{attribute 'qualified_only'}
VAR_GLOBAL
	Section 					: ARRAY[1..4] OF ST_Trip_Base;
	MasterStopPBPressed			: BOOL;
	CaseEStopCircuitBroken		: BOOL;
	ManualModeSelected			: BOOL;
	MCPLossDCpower				: BOOL;
	MCPsystemTripped			: BOOL;
	
	AnyEstopPressed 			: BOOL;
	AllDCpsuOK					: BOOL;
	AnyChargerOverTemp			: BOOL;
	AnyChargerLoadFault			: BOOL;
	AnyChargerInterlockOpen		: BOOL;
	AnyChargerFaulted			: BOOL; // same as summary fault
	//SystemTripped 				: BOOL;
	//InstrumentationFaulted		: BOOL;
	AnyChargeRlyFail			: BOOL;
	AnyDumpRlyFail				: BOOL;
	//AnyACInterlockFail			: BOOL;
	
	NoFaultDetected				: BOOL;
	ClearAllFaults				: BOOL;
END_VAR

(* stored: Version 1.1.0.1, ProductVersion 3.1.4024.11
   GVL Trips_DB: Id {b9292f11-9c83-43f6-9b30-6c69cf4aaa02} *)
